// Mitsubishi GX Works2 project: servo5   PLC: Q03UDV

PROGRAM MAIN
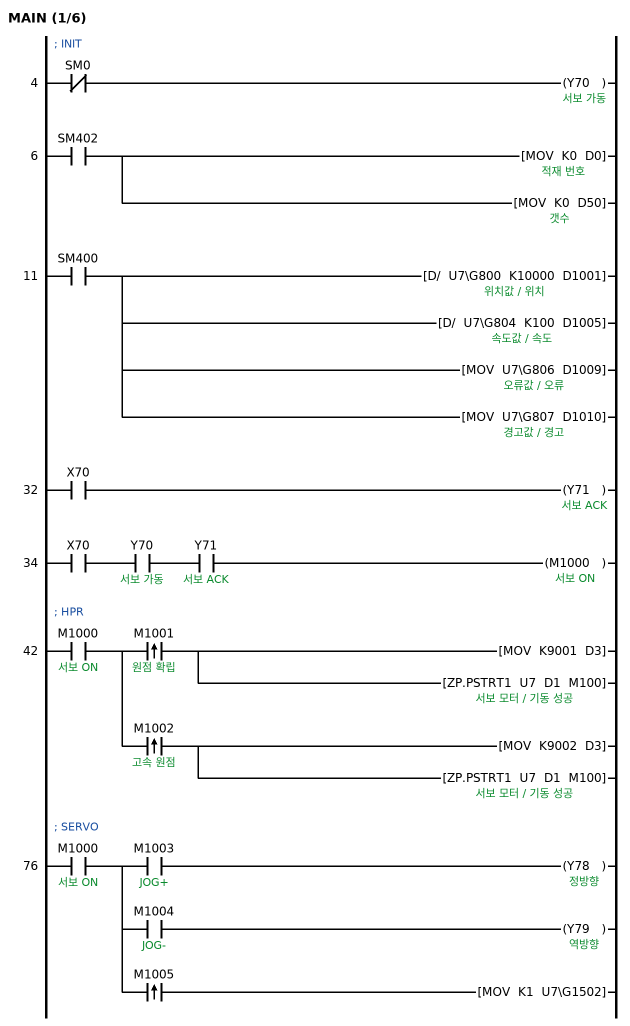
; INIT
4     LDI     SM0
      OUT     Y70  ; 서보 가동
6     LD      SM402
      MOV     K0 D0  ; 적재 번호
      MOV     K0 D50  ; 갯수
11    LD      SM400
      D/      U7\G800 K10000 D1001  ; 위치값 / 위치
      D/      U7\G804 K100 D1005  ; 속도값 / 속도
      MOV     U7\G806 D1009  ; 오류값 / 오류
      MOV     U7\G807 D1010  ; 경고값 / 경고
32    LD      X70
      OUT     Y71  ; 서보 ACK
34    LD      X70
      AND     Y70  ; 서보 가동
      AND     Y71  ; 서보 ACK
      OUT     M1000  ; 서보 ON
; HPR
42    LD      M1000  ; 서보 ON
      MPS
      ANDP    M1001  ; 원점 확립
      MOV     K9001 D3
      ZP.PSTRT1 U7 D1 M100  ; 서보 모터 / 기동 성공
      MPP
      ANDP    M1002  ; 고속 원점
      MOV     K9002 D3
      ZP.PSTRT1 U7 D1 M100
; SERVO
76    LD      M1000  ; 서보 ON
      MPS
      AND     M1003  ; JOG+
      OUT     Y78  ; 정방향
      MRD
      AND     M1004  ; JOG-
      OUT     Y79  ; 역방향
      MPP
      ANDP    M1005
      MOV     K1 U7\G1502
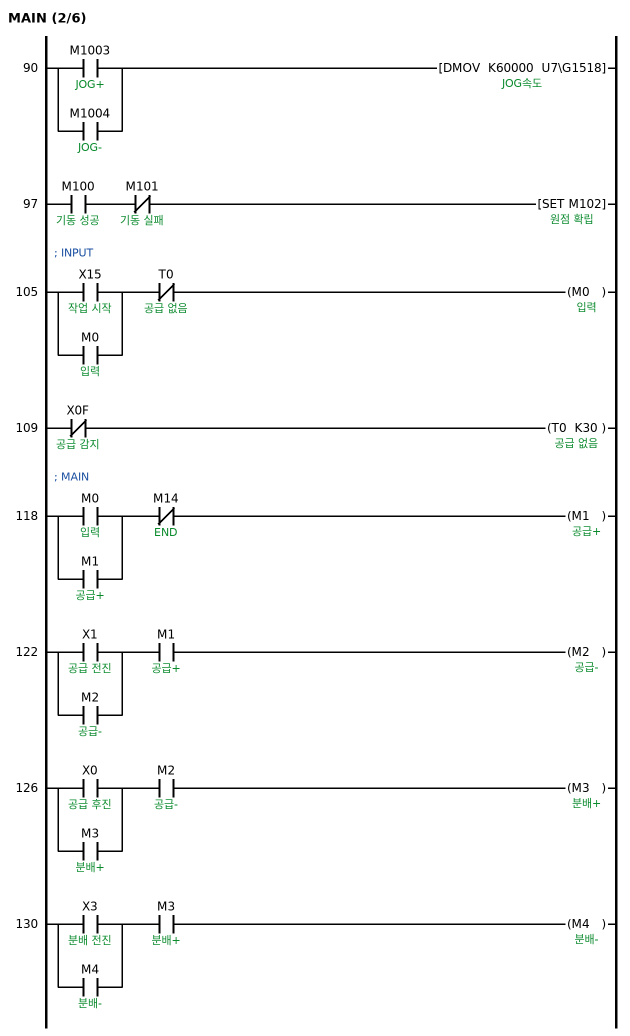
90    LD      M1003  ; JOG+
      OR      M1004  ; JOG-
      DMOV    K60000 U7\G1518  ; JOG속도
97    LD      M100  ; 기동 성공
      ANI     M101  ; 기동 실패
      SET     M102  ; 원점 확립
; INPUT
105   LD      X15  ; 작업 시작
      OR      M0  ; 입력
      ANI     T0  ; 공급 없음
      OUT     M0  ; 입력
109   LDI     X0F  ; 공급 감지
      OUT     T0 K30  ; 공급 없음
; MAIN
118   LD      M0  ; 입력
      OR      M1  ; 공급+
      ANI     M14  ; END
      OUT     M1  ; 공급+
122   LD      X1  ; 공급 전진
      OR      M2  ; 공급-
      AND     M1  ; 공급+
      OUT     M2  ; 공급-
126   LD      X0  ; 공급 후진
      OR      M3  ; 분배+
      AND     M2  ; 공급-
      OUT     M3  ; 분배+
130   LD      X3  ; 분배 전진
      OR      M4  ; 분배-
      AND     M3  ; 분배+
      OUT     M4  ; 분배-
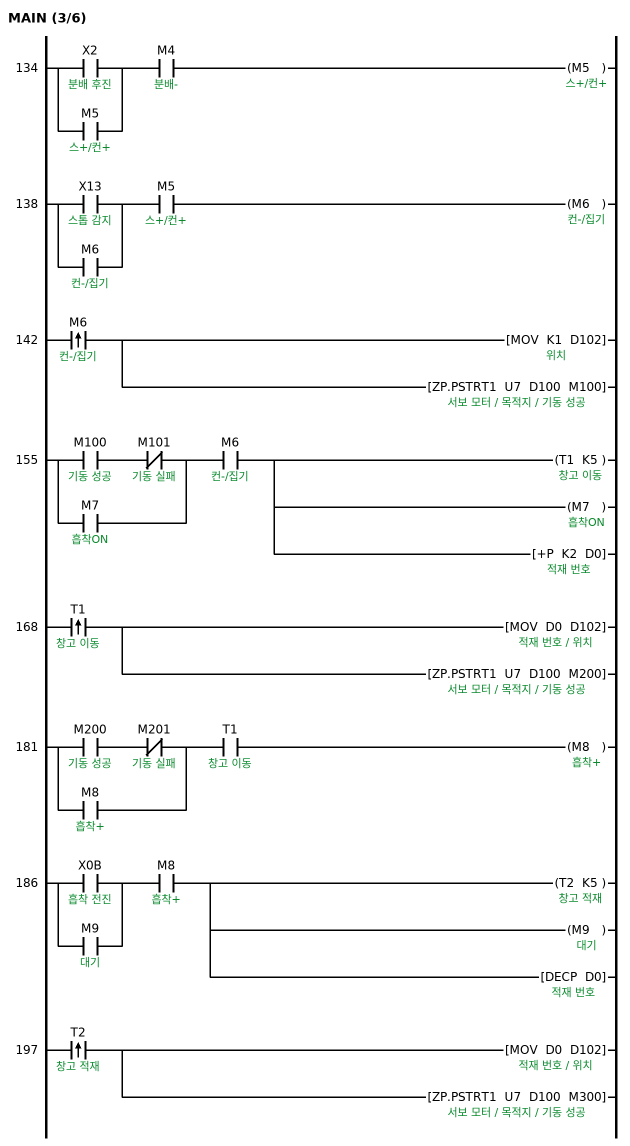
134   LD      X2  ; 분배 후진
      OR      M5  ; 스+/컨+
      AND     M4  ; 분배-
      OUT     M5  ; 스+/컨+
138   LD      X13  ; 스톱 감지
      OR      M6  ; 컨-/집기
      AND     M5  ; 스+/컨+
      OUT     M6  ; 컨-/집기
142   LDP     M6  ; 컨-/집기
      MOV     K1 D102  ; 위치
      ZP.PSTRT1 U7 D100 M100  ; 목적지
155   LD      M100  ; 기동 성공
      ANI     M101  ; 기동 실패
      OR      M7  ; 흡착ON
      AND     M6  ; 컨-/집기
      OUT     T1 K5  ; 창고 이동
      OUT     M7  ; 흡착ON
      +P      K2 D0
168   LDP     T1  ; 창고 이동
      MOV     D0 D102
      ZP.PSTRT1 U7 D100 M200  ; 기동 성공
181   LD      M200  ; 기동 성공
      ANI     M201  ; 기동 실패
      OR      M8  ; 흡착+
      AND     T1  ; 창고 이동
      OUT     M8  ; 흡착+
186   LD      X0B  ; 흡착 전진
      OR      M9  ; 대기
      AND     M8  ; 흡착+
      OUT     T2 K5  ; 창고 적재
      OUT     M9  ; 대기
      DECP    D0
197   LDP     T2  ; 창고 적재
      MOV     D0 D102
      ZP.PSTRT1 U7 D100 M300  ; 기동 성공
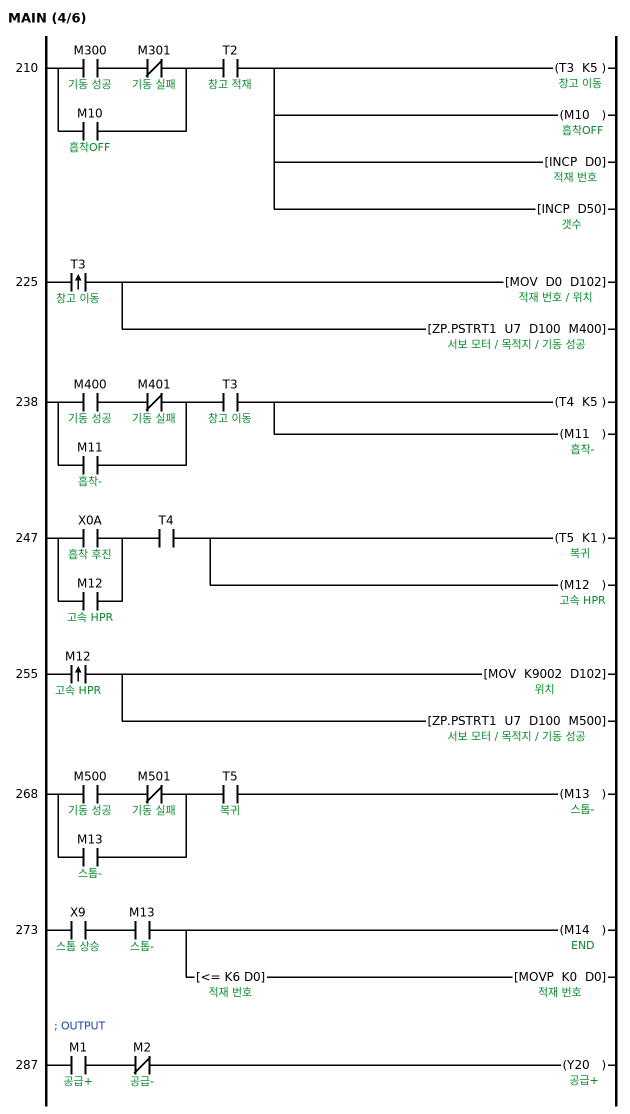
210   LD      M300  ; 기동 성공
      ANI     M301  ; 기동 실패
      OR      M10  ; 흡착OFF
      AND     T2  ; 창고 적재
      OUT     T3 K5  ; 창고 이동
      OUT     M10  ; 흡착OFF
      INCP    D0
      INCP    D50
225   LDP     T3  ; 창고 이동
      MOV     D0 D102
      ZP.PSTRT1 U7 D100 M400  ; 기동 성공
238   LD      M400  ; 기동 성공
      ANI     M401  ; 기동 실패
      OR      M11  ; 흡착-
      AND     T3  ; 창고 이동
      OUT     T4 K5
      OUT     M11  ; 흡착-
247   LD      X0A  ; 흡착 후진
      OR      M12  ; 고속 HPR
      AND     T4
      OUT     T5 K1  ; 복귀
      OUT     M12  ; 고속 HPR
255   LDP     M12  ; 고속 HPR
      MOV     K9002 D102
      ZP.PSTRT1 U7 D100 M500  ; 기동 성공
268   LD      M500  ; 기동 성공
      ANI     M501  ; 기동 실패
      OR      M13  ; 스톱-
      AND     T5  ; 복귀
      OUT     M13  ; 스톱-
273   LD      X9  ; 스톱 상승
      AND     M13  ; 스톱-
      OUT     M14  ; END
      AND<=   K6 D0  ; 적재 번호
      MOVP    K0 D0
; OUTPUT
287   LD      M1  ; 공급+
      ANI     M2  ; 공급-
      OUT     Y20  ; 공급+
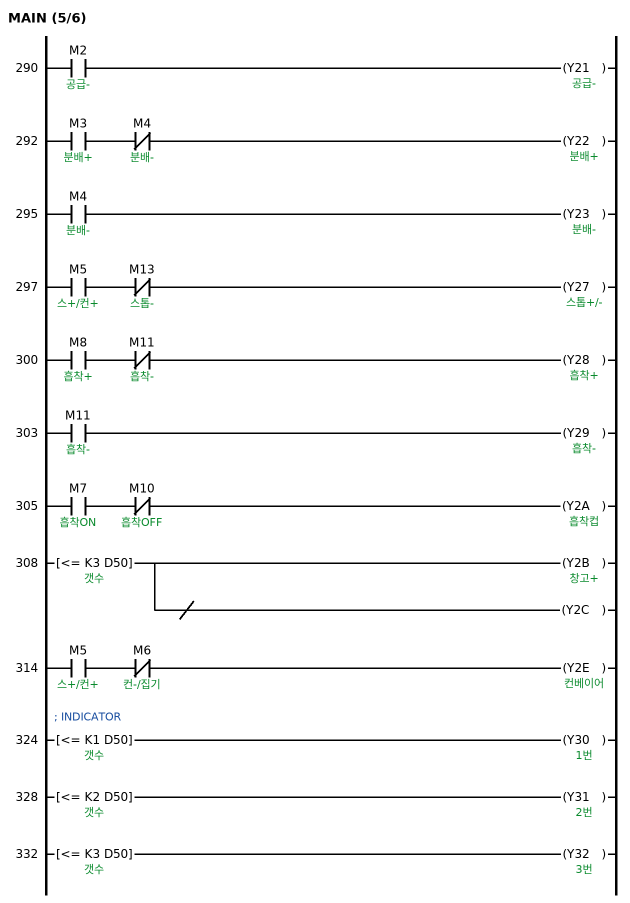
290   LD      M2  ; 공급-
      OUT     Y21  ; 공급-
292   LD      M3  ; 분배+
      ANI     M4  ; 분배-
      OUT     Y22  ; 분배+
295   LD      M4  ; 분배-
      OUT     Y23  ; 분배-
297   LD      M5  ; 스+/컨+
      ANI     M13  ; 스톱-
      OUT     Y27  ; 스톱+/-
300   LD      M8  ; 흡착+
      ANI     M11  ; 흡착-
      OUT     Y28  ; 흡착+
303   LD      M11  ; 흡착-
      OUT     Y29  ; 흡착-
305   LD      M7  ; 흡착ON
      ANI     M10  ; 흡착OFF
      OUT     Y2A  ; 흡착컵
308   LD<=    K3 D50  ; 갯수
      OUT     Y2B  ; 창고+
      INV
      OUT     Y2C
314   LD      M5  ; 스+/컨+
      ANI     M6  ; 컨-/집기
      OUT     Y2E  ; 컨베이어
; INDICATOR
324   LD<=    K1 D50  ; 갯수
      OUT     Y30  ; 1번
328   LD<=    K2 D50  ; 갯수
      OUT     Y31  ; 2번
332   LD<=    K3 D50  ; 갯수
      OUT     Y32  ; 3번
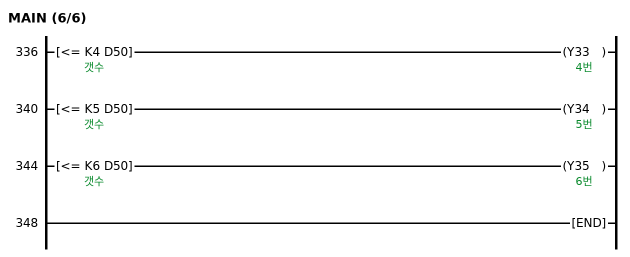
336   LD<=    K4 D50  ; 갯수
      OUT     Y33  ; 4번
340   LD<=    K5 D50  ; 갯수
      OUT     Y34  ; 5번
344   LD<=    K6 D50  ; 갯수
      OUT     Y35  ; 6번
348   END
END_PROGRAM

// device comments not shown above
X8  ; 스톱 상승
M600  ; 기동 성공
M601  ; 기동 실패
D2  ; 몫
D10010  ; 경고
